NAMESPACE LineA1
ORGANIZATION_BLOCK Main_LineA1
TITLE = "Main Program Sweep (Cycle)"
{ S7_Optimized_Access := 'TRUE' ; Published := 'FALSE' }
VERSION : 0.1

BEGIN
	IDB_LineA1();

END_ORGANIZATION_BLOCK
END_NAMESPACE

